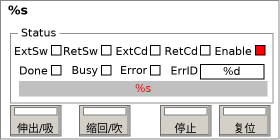
VISUALIZATION cylinderModuleVisu  // 280x140
VAR_IN_OUT
	userData: CylinderModuleHMI;
END_VAR
    Button (10,105 51x31), "伸出/吸", input disabled if: NOT userData.HMIEnable
        tap userData.extend
    Rectangle (14,107 43x8), colour toggle: userData.extRelay
    GroupBox (10,25 263x78), "Status"
        Label (54,20 37x13), "RetSw"
        Label (4,20 37x13), "ExtSw"
        RoundedRectangle (41,20 10x10), colour toggle: userData.extAprSw
        RoundedRectangle (91,20 10x10), colour toggle: userData.retAprSw
        RoundedRectangle (41,40 10x10), colour toggle: userData.done
        RoundedRectangle (245,20 10x10), colour toggle: userData.enable
        RoundedRectangle (91,40 10x10), colour toggle: userData.busy
        RoundedRectangle (140,40 10x10), colour toggle: userData.error
        Rectangle (190,39 64x15), "%d", text variable: userData.errID
        Label (104,20 37x13), "ExtCd"
        RoundedRectangle (140,20 10x10), colour toggle: userData.extcondition
        Label (154,20 37x13), "RetCd"
        RoundedRectangle (190,20 10x10), colour toggle: userData.retcondition
        Rectangle (9,56 248x15), "%s", text variable: userData.errTXT
        Label (206,20 39x13), "Enable"
        Label (158,39 33x14), "ErrID"
        Label (110,39 30x13), "Error"
        Label (61,39 30x13), "Busy"
        Label (8,38 33x16), "Done"
    Button (79,105 51x31), "缩回/吹", input disabled if: NOT userData.HMIEnable
        tap userData.retract
    Rectangle (83,107 43x8), colour toggle: userData.retRelay
    Button (219,105 51x31), "复位"
        tap userData.reset
    Rectangle (223,107 43x8), colour toggle: userData.error
    Rectangle (5,0 267x20), "%s", text variable: userData.nameTXT
    Button (160,105 51x31), "停止"
        tap userData.stop
    Rectangle (164,107 43x8)
END_VISUALIZATION

(* stored: Version 1.1.0.1, ProductVersion 3.1.4024.4
   Visu cylinderModuleVisu: Id {68cce8c2-2e88-4a95-b5f9-f6047c373237} *)
